// TIA Portal project "LinkedList_v000_000_001" (V16)

(* hardware
DEVICE "S7-1200 station_1"  S7-1200 Station
   slot 0: "Rack_0"  S7-1200 Rack  Rack  V1.0
   slot 1: "PLC_1"  CPU 1212C DC/DC/DC  6ES7 212-1AE40-0XB0  V4.4
*)

// ===== PLC "PLC_1"  CPU 1212C DC/DC/DC =====

VAR_GLOBAL   // PLC tag table "Default tag table"
   "System_Byte" AT %MB1 : Byte;
   "FirstScan" AT %M1.0 : Bool;
   "DiagStatusUpdate" AT %M1.1 : Bool;
   "AlwaysTRUE" AT %M1.2 : Bool;
   "AlwaysFALSE" AT %M1.3 : Bool;
   "Clock_Byte" AT %MB0 : Byte;
   "Clock_10Hz" AT %M0.0 : Bool;
   "Clock_5Hz" AT %M0.1 : Bool;
   "Clock_2.5Hz" AT %M0.2 : Bool;
   "Clock_2Hz" AT %M0.3 : Bool;
   "Clock_1.25Hz" AT %M0.4 : Bool;
   "Clock_1Hz" AT %M0.5 : Bool;
   "Clock_0.625Hz" AT %M0.6 : Bool;
   "Clock_0.5Hz" AT %M0.7 : Bool;
END_VAR

TYPE "LinkedList.Node.Payload.UDT"
   STRUCT
      id : Char;
      status : String;
   END_STRUCT;
END_TYPE

TYPE "LinkedList.Node.UDT"
   STRUCT
      data : "LinkedList.Node.Payload.UDT";
      pointer : DInt;
   END_STRUCT;
END_TYPE

TYPE "LinkedList.UDT"
   STRUCT
      head : DInt;
      list : Array[0..4] of "LinkedList.Node.UDT";
   END_STRUCT;
END_TYPE

FUNCTION_BLOCK "LinkedList"   // FB1, SCL
TITLE = Linked List
{ S7_Optimized_Access := 'TRUE' }
AUTHOR : Machado
FAMILY : LinkedList
VERSION : 0.1
   VAR
      list : "LinkedList.UDT";
   END_VAR
BEGIN
   #list.list[0].data.id;
END_FUNCTION_BLOCK

ORGANIZATION_BLOCK "Main"   // OB1, LAD, ProgramCycle
TITLE = "Main Program Sweep (Cycle)"
{ S7_Optimized_Access := 'TRUE' }
VERSION : 0.1
   VAR_INPUT
      Initial_Call : Bool;   // Initial call of this OB
      Remanence : Bool;   // =True, if remanent data are available
   END_VAR
BEGIN
END_ORGANIZATION_BLOCK